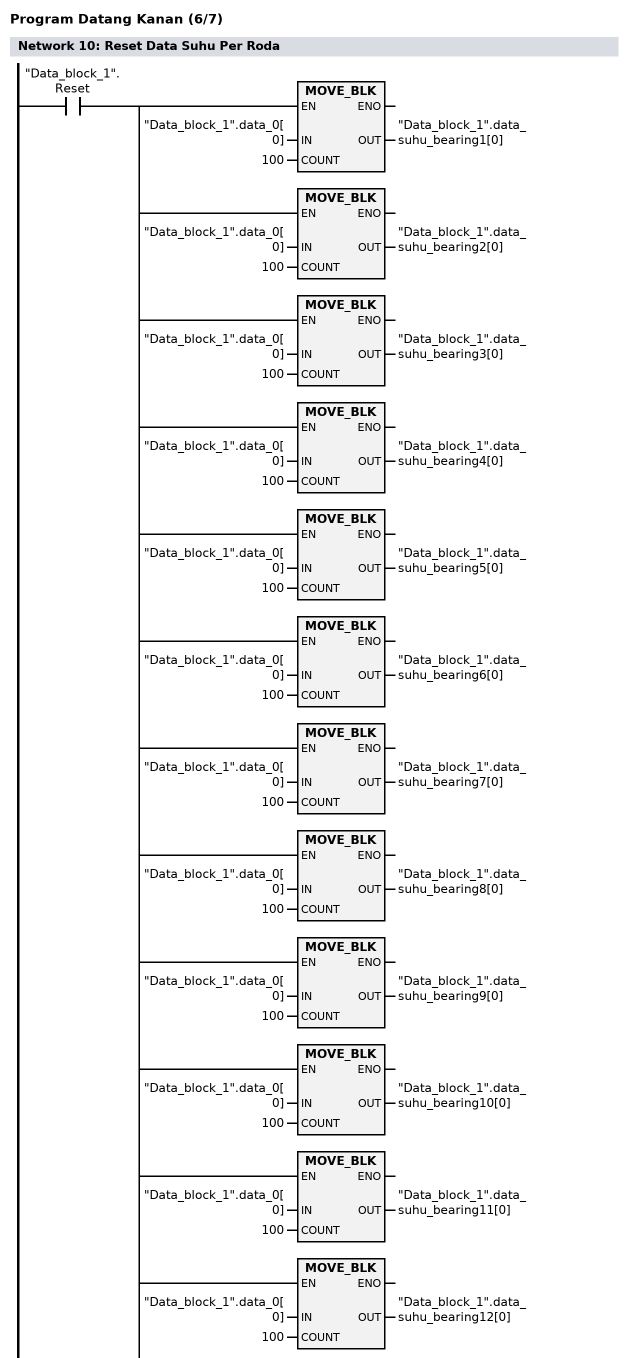
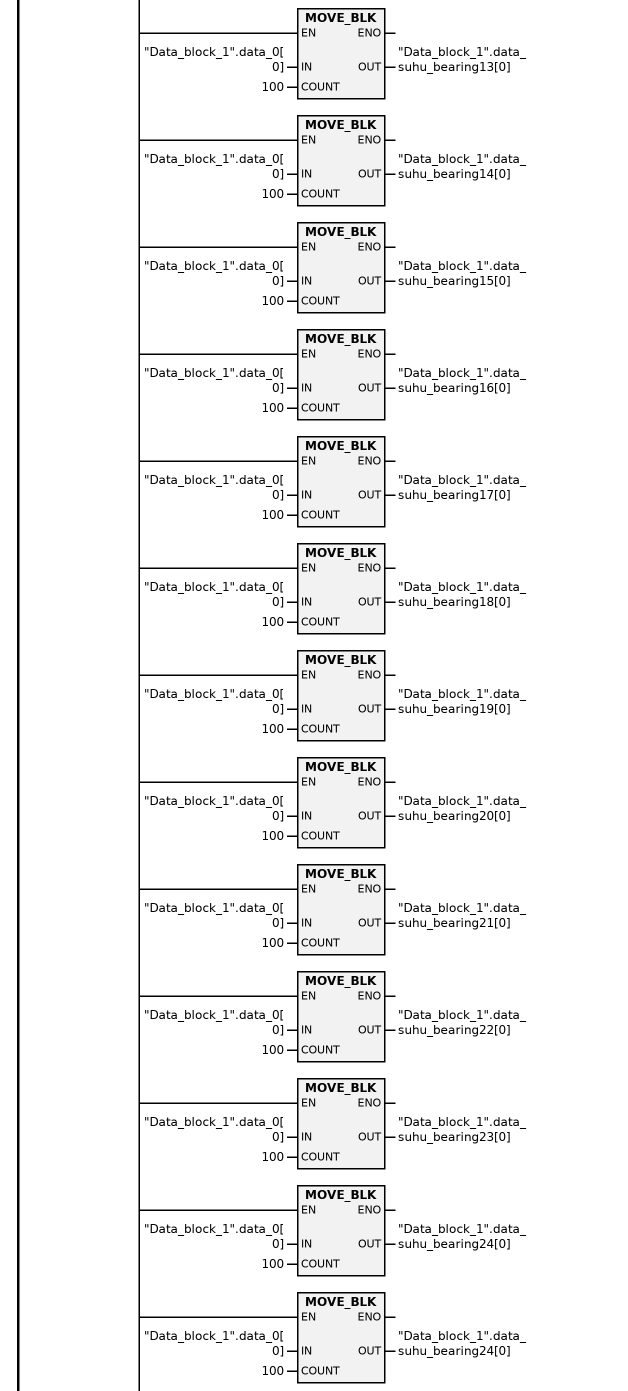
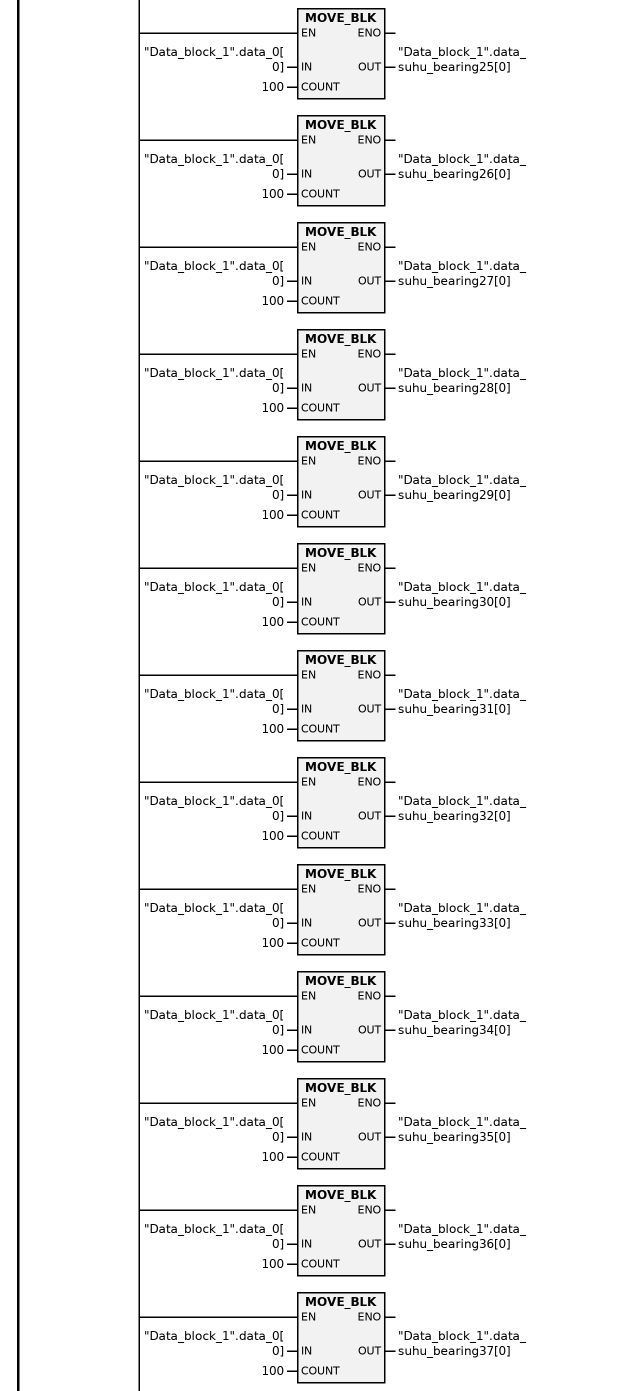
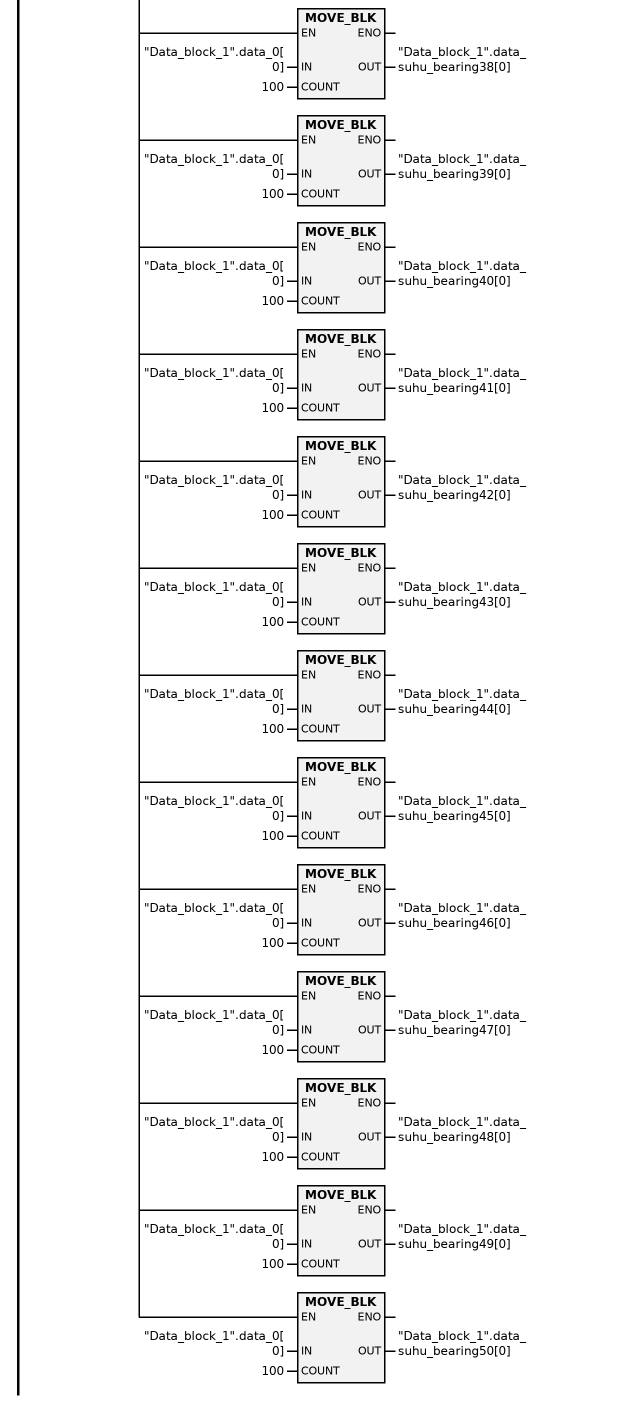
   #_w1 := "Data_block_1".Reset;
   IF #_w1 THEN
       MOVE_BLK(IN := "Data_block_1".data_0[0], COUNT := 100, OUT => "Data_block_1".data_suhu_bearing1[0]);
       MOVE_BLK(IN := "Data_block_1".data_0[0], COUNT := 100, OUT => "Data_block_1".data_suhu_bearing2[0]);
       MOVE_BLK(IN := "Data_block_1".data_0[0], COUNT := 100, OUT => "Data_block_1".data_suhu_bearing3[0]);
       MOVE_BLK(IN := "Data_block_1".data_0[0], COUNT := 100, OUT => "Data_block_1".data_suhu_bearing4[0]);
       MOVE_BLK(IN := "Data_block_1".data_0[0], COUNT := 100, OUT => "Data_block_1".data_suhu_bearing5[0]);
       MOVE_BLK(IN := "Data_block_1".data_0[0], COUNT := 100, OUT => "Data_block_1".data_suhu_bearing6[0]);
       MOVE_BLK(IN := "Data_block_1".data_0[0], COUNT := 100, OUT => "Data_block_1".data_suhu_bearing7[0]);
       MOVE_BLK(IN := "Data_block_1".data_0[0], COUNT := 100, OUT => "Data_block_1".data_suhu_bearing8[0]);
       MOVE_BLK(IN := "Data_block_1".data_0[0], COUNT := 100, OUT => "Data_block_1".data_suhu_bearing9[0]);
       MOVE_BLK(IN := "Data_block_1".data_0[0], COUNT := 100, OUT => "Data_block_1".data_suhu_bearing10[0]);
       MOVE_BLK(IN := "Data_block_1".data_0[0], COUNT := 100, OUT => "Data_block_1".data_suhu_bearing11[0]);
       MOVE_BLK(IN := "Data_block_1".data_0[0], COUNT := 100, OUT => "Data_block_1".data_suhu_bearing12[0]);
       MOVE_BLK(IN := "Data_block_1".data_0[0], COUNT := 100, OUT => "Data_block_1".data_suhu_bearing13[0]);
       MOVE_BLK(IN := "Data_block_1".data_0[0], COUNT := 100, OUT => "Data_block_1".data_suhu_bearing14[0]);
       MOVE_BLK(IN := "Data_block_1".data_0[0], COUNT := 100, OUT => "Data_block_1".data_suhu_bearing15[0]);
       MOVE_BLK(IN := "Data_block_1".data_0[0], COUNT := 100, OUT => "Data_block_1".data_suhu_bearing16[0]);
       MOVE_BLK(IN := "Data_block_1".data_0[0], COUNT := 100, OUT => "Data_block_1".data_suhu_bearing17[0]);
       MOVE_BLK(IN := "Data_block_1".data_0[0], COUNT := 100, OUT => "Data_block_1".data_suhu_bearing18[0]);
       MOVE_BLK(IN := "Data_block_1".data_0[0], COUNT := 100, OUT => "Data_block_1".data_suhu_bearing19[0]);
       MOVE_BLK(IN := "Data_block_1".data_0[0], COUNT := 100, OUT => "Data_block_1".data_suhu_bearing20[0]);
       MOVE_BLK(IN := "Data_block_1".data_0[0], COUNT := 100, OUT => "Data_block_1".data_suhu_bearing21[0]);
       MOVE_BLK(IN := "Data_block_1".data_0[0], COUNT := 100, OUT => "Data_block_1".data_suhu_bearing22[0]);
       MOVE_BLK(IN := "Data_block_1".data_0[0], COUNT := 100, OUT => "Data_block_1".data_suhu_bearing23[0]);
       MOVE_BLK(IN := "Data_block_1".data_0[0], COUNT := 100, OUT => "Data_block_1".data_suhu_bearing24[0]);
       MOVE_BLK(IN := "Data_block_1".data_0[0], COUNT := 100, OUT => "Data_block_1".data_suhu_bearing24[0]);
       MOVE_BLK(IN := "Data_block_1".data_0[0], COUNT := 100, OUT => "Data_block_1".data_suhu_bearing25[0]);
       MOVE_BLK(IN := "Data_block_1".data_0[0], COUNT := 100, OUT => "Data_block_1".data_suhu_bearing26[0]);
       MOVE_BLK(IN := "Data_block_1".data_0[0], COUNT := 100, OUT => "Data_block_1".data_suhu_bearing27[0]);
       MOVE_BLK(IN := "Data_block_1".data_0[0], COUNT := 100, OUT => "Data_block_1".data_suhu_bearing28[0]);
       MOVE_BLK(IN := "Data_block_1".data_0[0], COUNT := 100, OUT => "Data_block_1".data_suhu_bearing29[0]);
       MOVE_BLK(IN := "Data_block_1".data_0[0], COUNT := 100, OUT => "Data_block_1".data_suhu_bearing30[0]);
       MOVE_BLK(IN := "Data_block_1".data_0[0], COUNT := 100, OUT => "Data_block_1".data_suhu_bearing31[0]);
       MOVE_BLK(IN := "Data_block_1".data_0[0], COUNT := 100, OUT => "Data_block_1".data_suhu_bearing32[0]);
       MOVE_BLK(IN := "Data_block_1".data_0[0], COUNT := 100, OUT => "Data_block_1".data_suhu_bearing33[0]);
       MOVE_BLK(IN := "Data_block_1".data_0[0], COUNT := 100, OUT => "Data_block_1".data_suhu_bearing34[0]);
       MOVE_BLK(IN := "Data_block_1".data_0[0], COUNT := 100, OUT => "Data_block_1".data_suhu_bearing35[0]);
       MOVE_BLK(IN := "Data_block_1".data_0[0], COUNT := 100, OUT => "Data_block_1".data_suhu_bearing36[0]);
       MOVE_BLK(IN := "Data_block_1".data_0[0], COUNT := 100, OUT => "Data_block_1".data_suhu_bearing37[0]);
       MOVE_BLK(IN := "Data_block_1".data_0[0], COUNT := 100, OUT => "Data_block_1".data_suhu_bearing38[0]);
       MOVE_BLK(IN := "Data_block_1".data_0[0], COUNT := 100, OUT => "Data_block_1".data_suhu_bearing39[0]);
       MOVE_BLK(IN := "Data_block_1".data_0[0], COUNT := 100, OUT => "Data_block_1".data_suhu_bearing40[0]);
       MOVE_BLK(IN := "Data_block_1".data_0[0], COUNT := 100, OUT => "Data_block_1".data_suhu_bearing41[0]);
       MOVE_BLK(IN := "Data_block_1".data_0[0], COUNT := 100, OUT => "Data_block_1".data_suhu_bearing42[0]);
       MOVE_BLK(IN := "Data_block_1".data_0[0], COUNT := 100, OUT => "Data_block_1".data_suhu_bearing43[0]);
       MOVE_BLK(IN := "Data_block_1".data_0[0], COUNT := 100, OUT => "Data_block_1".data_suhu_bearing44[0]);
       MOVE_BLK(IN := "Data_block_1".data_0[0], COUNT := 100, OUT => "Data_block_1".data_suhu_bearing45[0]);
       MOVE_BLK(IN := "Data_block_1".data_0[0], COUNT := 100, OUT => "Data_block_1".data_suhu_bearing46[0]);
       MOVE_BLK(IN := "Data_block_1".data_0[0], COUNT := 100, OUT => "Data_block_1".data_suhu_bearing47[0]);
       MOVE_BLK(IN := "Data_block_1".data_0[0], COUNT := 100, OUT => "Data_block_1".data_suhu_bearing48[0]);
       MOVE_BLK(IN := "Data_block_1".data_0[0], COUNT := 100, OUT => "Data_block_1".data_suhu_bearing49[0]);
       MOVE_BLK(IN := "Data_block_1".data_0[0], COUNT := 100, OUT => "Data_block_1".data_suhu_bearing50[0]);
   END_IF;
END_REGION

REGION Network 11
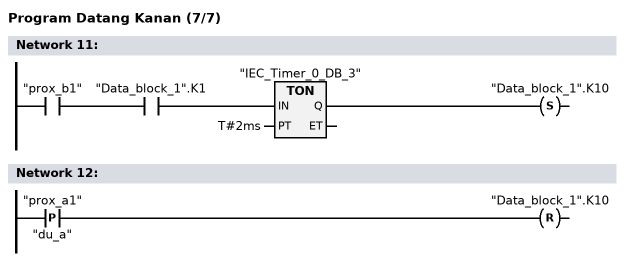
   "IEC_Timer_0_DB_3".TON(IN := "prox_b1" AND "Data_block_1".K1, PT := T#2ms);
   IF "IEC_Timer_0_DB_3".Q THEN "Data_block_1".K10 := TRUE; END_IF;
END_REGION

REGION Network 12
   RUNG wire#powerrail
      P_Contact(operand := "prox_a1", bit := "du_a")
      R_Coil( "Data_block_1".K10 )
   END_RUNG
   // the same network as SCL:
   #_w1 := "prox_a1" AND NOT "du_a";   // rising edge of "prox_a1"
   "du_a" := "prox_a1";
   IF #_w1 THEN "Data_block_1".K10 := FALSE; END_IF;
END_REGION
END_ORGANIZATION_BLOCK

ORGANIZATION_BLOCK "Program General"   // OB124, LAD, ProgramCycle
TITLE = General
{ S7_Optimized_Access := 'TRUE' }
VERSION : 0.1
   VAR_INPUT
      Initial_Call : Bool;   // Initial call of this OB
      Remanence : Bool;   // =True, if remanent data are available
   END_VAR
   VAR_TEMP   // added for the SCL form of the ladder/FBD networks
      _w1 : Bool;
   END_VAR
BEGIN

REGION Network 1: Counter sensor
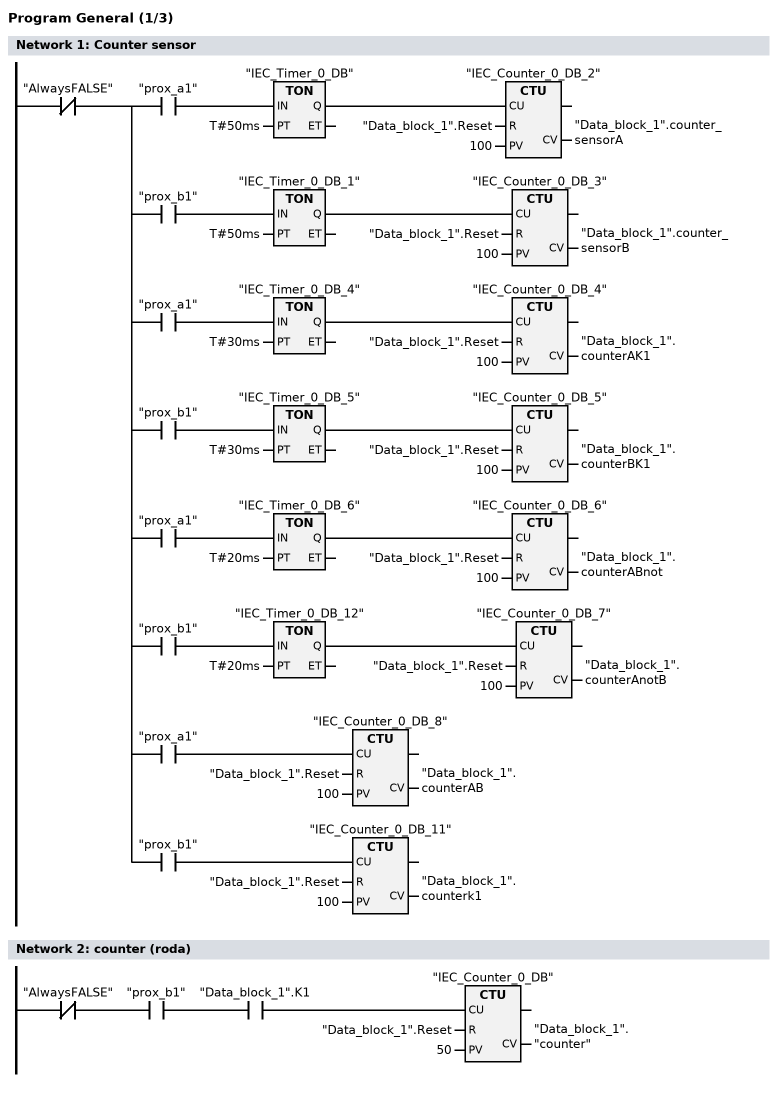
   "IEC_Timer_0_DB".TON(IN := NOT "AlwaysFALSE" AND "prox_a1", PT := T#50ms);
   "IEC_Counter_0_DB_2".CTU(CU := "IEC_Timer_0_DB".Q,
                           R := "Data_block_1".Reset,
                           PV := 100,
                           CV => "Data_block_1".counter_sensorA);
   "IEC_Timer_0_DB_1".TON(IN := NOT "AlwaysFALSE" AND "prox_b1", PT := T#50ms);
   "IEC_Counter_0_DB_3".CTU(CU := "IEC_Timer_0_DB_1".Q,
                           R := "Data_block_1".Reset,
                           PV := 100,
                           CV => "Data_block_1".counter_sensorB);
   "IEC_Timer_0_DB_4".TON(IN := NOT "AlwaysFALSE" AND "prox_a1", PT := T#30ms);
   "IEC_Counter_0_DB_4".CTU(CU := "IEC_Timer_0_DB_4".Q,
                           R := "Data_block_1".Reset,
                           PV := 100,
                           CV => "Data_block_1".counterAK1);
   "IEC_Timer_0_DB_5".TON(IN := NOT "AlwaysFALSE" AND "prox_b1", PT := T#30ms);
   "IEC_Counter_0_DB_5".CTU(CU := "IEC_Timer_0_DB_5".Q,
                           R := "Data_block_1".Reset,
                           PV := 100,
                           CV => "Data_block_1".counterBK1);
   "IEC_Timer_0_DB_6".TON(IN := NOT "AlwaysFALSE" AND "prox_a1", PT := T#20ms);
   "IEC_Counter_0_DB_6".CTU(CU := "IEC_Timer_0_DB_6".Q,
                           R := "Data_block_1".Reset,
                           PV := 100,
                           CV => "Data_block_1".counterABnot);
   "IEC_Timer_0_DB_12".TON(IN := NOT "AlwaysFALSE" AND "prox_b1", PT := T#20ms);
   "IEC_Counter_0_DB_7".CTU(CU := "IEC_Timer_0_DB_12".Q,
                           R := "Data_block_1".Reset,
                           PV := 100,
                           CV => "Data_block_1".counterAnotB);
   "IEC_Counter_0_DB_8".CTU(CU := NOT "AlwaysFALSE" AND "prox_a1",
                           R := "Data_block_1".Reset,
                           PV := 100,
                           CV => "Data_block_1".counterAB);
   "IEC_Counter_0_DB_11".CTU(CU := NOT "AlwaysFALSE" AND "prox_b1",
                           R := "Data_block_1".Reset,
                           PV := 100,
                           CV => "Data_block_1".counterk1);
END_REGION

REGION Network 2: counter (roda)
   "IEC_Counter_0_DB".CTU(CU := NOT "AlwaysFALSE" AND "prox_b1" AND "Data_block_1".K1,
                          R := "Data_block_1".Reset,
                          PV := 50,
                          CV => "Data_block_1"."counter");
END_REGION

REGION Network 3: Timer Mengukur kecepatan kereta
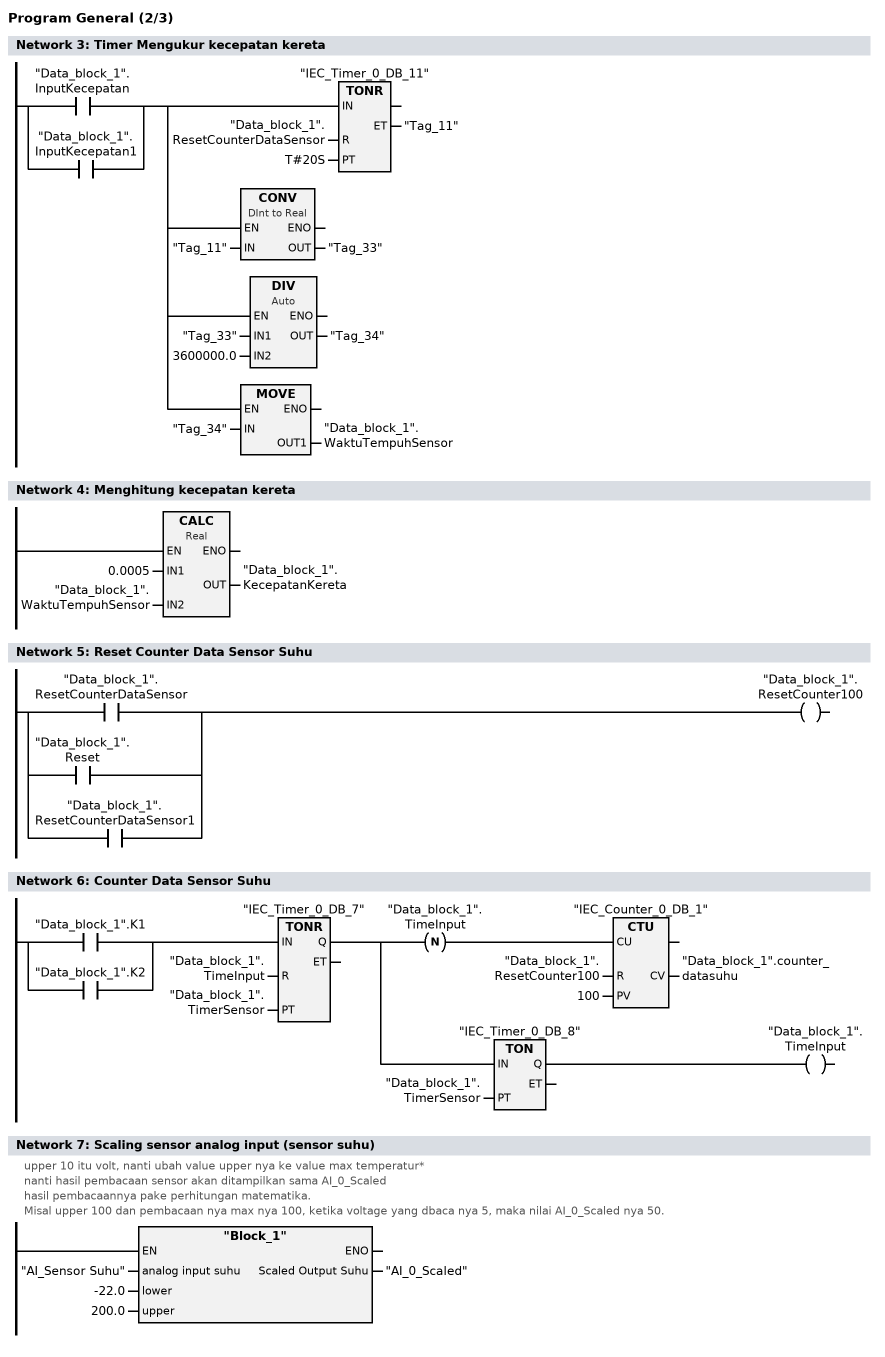
   #_w1 := "Data_block_1".InputKecepatan OR "Data_block_1".InputKecepatan1;
   "IEC_Timer_0_DB_11".TONR(IN := #_w1, R := "Data_block_1".ResetCounterDataSensor, PT := T#20S, ET => "Tag_11");
   IF #_w1 THEN
       "Tag_33" := DINT_TO_REAL("Tag_11");
       "Tag_34" := "Tag_33" / 3600000.0;
       "Data_block_1".WaktuTempuhSensor := "Tag_34";
   END_IF;
END_REGION

REGION Network 4: Menghitung kecepatan kereta
   CALC(in1 := 0.0005, in2 := "Data_block_1".WaktuTempuhSensor, out => "Data_block_1".KecepatanKereta);
END_REGION

REGION Network 5: Reset Counter Data Sensor Suhu
   RUNG wire#powerrail
      Contact( "Data_block_1".ResetCounterDataSensor )
      wire#w1
      Coil( "Data_block_1".ResetCounter100 )
   END_RUNG
   RUNG wire#powerrail
      Contact( "Data_block_1".Reset )
   END_RUNG wire#w1
   RUNG wire#powerrail
      Contact( "Data_block_1".ResetCounterDataSensor1 )
   END_RUNG wire#w1
   // the same network as SCL:
   "Data_block_1".ResetCounter100 := "Data_block_1".ResetCounterDataSensor OR "Data_block_1".Reset OR "Data_block_1".ResetCounterDataSensor1;
END_REGION

REGION Network 6: Counter Data Sensor Suhu
   "IEC_Timer_0_DB_7".TONR(IN := "Data_block_1".K1 OR "Data_block_1".K2,
                           R := "Data_block_1".TimeInput,
                           PT := "Data_block_1".TimerSensor);
   #_w1 := NOT "IEC_Timer_0_DB_7".Q AND "Data_block_1".TimeInput;   // falling edge
   "Data_block_1".TimeInput := "IEC_Timer_0_DB_7".Q;
   "IEC_Counter_0_DB_1".CTU(CU := #_w1,
                           R := "Data_block_1".ResetCounter100,
                           PV := 100,
                           CV => "Data_block_1".counter_datasuhu);
   "IEC_Timer_0_DB_8".TON(IN := "IEC_Timer_0_DB_7".Q, PT := "Data_block_1".TimerSensor);
   "Data_block_1".TimeInput := "IEC_Timer_0_DB_8".Q;
END_REGION

REGION Network 7: Scaling sensor analog input (sensor suhu)
   // upper 10 itu volt, nanti ubah value upper nya ke value max temperatur* 
   // nanti hasil pembacaan sensor akan ditampilkan sama AI_0_Scaled
   // hasil pembacaannya pake perhitungan matematika. 
   // Misal upper 100 dan pembacaan nya max nya 100, ketika voltage yang dbaca nya 5, maka nilai AI_0_Scaled nya 50.
   RUNG wire#powerrail
      "Block_1"("analog input suhu" := "AI_Sensor Suhu", lower := -22.0, upper := 200.0, "Scaled Output Suhu" => "AI_0_Scaled")
   END_RUNG
   // the same network as SCL:
   "Block_1"("analog input suhu" := "AI_Sensor Suhu",
             lower := -22.0,
             upper := 200.0,
             "Scaled Output Suhu" => "AI_0_Scaled");
END_REGION

REGION Network 8: Data memory suhu kanan
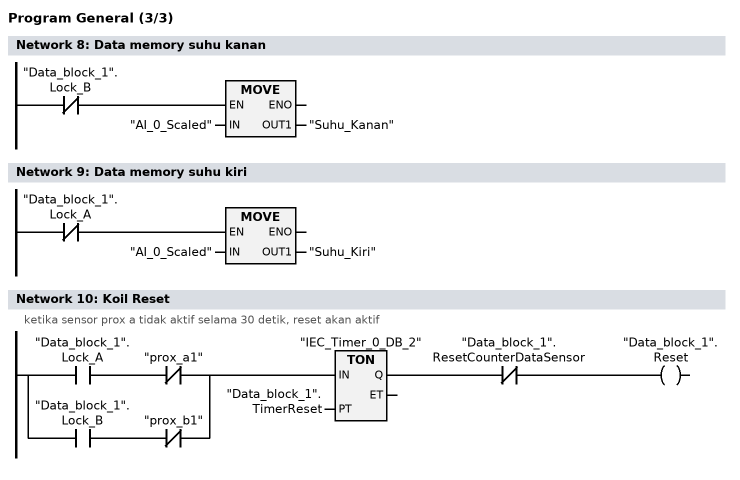
   RUNG wire#powerrail
      I_Contact( "Data_block_1".Lock_B )
      Move(in := "AI_0_Scaled", out1 => "Suhu_Kanan")
   END_RUNG
   // the same network as SCL:
   IF NOT "Data_block_1".Lock_B THEN "Suhu_Kanan" := "AI_0_Scaled"; END_IF;
END_REGION

REGION Network 9: Data memory suhu kiri
   RUNG wire#powerrail
      I_Contact( "Data_block_1".Lock_A )
      Move(in := "AI_0_Scaled", out1 => "Suhu_Kiri")
   END_RUNG
   // the same network as SCL:
   IF NOT "Data_block_1".Lock_A THEN "Suhu_Kiri" := "AI_0_Scaled"; END_IF;
END_REGION

REGION Network 10: Koil Reset
   // ketika sensor prox a tidak aktif selama 30 detik, reset akan aktif
   "IEC_Timer_0_DB_2".TON(IN := ("Data_block_1".Lock_A AND NOT "prox_a1") OR ("Data_block_1".Lock_B AND NOT "prox_b1"),
                          PT := "Data_block_1".TimerReset);
   "Data_block_1".Reset := "IEC_Timer_0_DB_2".Q AND NOT "Data_block_1".ResetCounterDataSensor;
END_REGION
END_ORGANIZATION_BLOCK

(* ===== HMI "HMI_RT_1" =====
system functions are stored by id; their names below are inferred from use
connection "Connection_1": ETHERNET, S7_1200_OMS
connection "HMI_Connection_1": ETHERNET, S7_1200_OMS

HMI tags "Default tag table"
   "prox_a" : Bool = PLC prox_a1 AT %I0.0, 1 s
   "prox_b" : Bool = PLC prox_b1 AT %I0.1, 1 s
   "Q1" : Bool = PLC "Q1-1" AT %M0.0, 1 s
   "Q2" : Bool = PLC "Q2-1" AT %M0.1, 1 s
   "du_a" : Bool = PLC du_a AT %M0.2, 1 s
   "dd_b" : Bool = PLC dd_b AT %M0.3, 1 s
   "k_proxa" : Bool = PLC k_proxa AT %M0.4, 1 s
   "k_proxb" : Bool = PLC k_proxb AT %M0.5, 1 s
   "counter" : Bool = PLC counter AT %M0.6, 1 s
   "pemutus" : Bool = PLC pemutus AT %M0.7, 1 s
   "du_b" : Bool = PLC "ProxA+" AT %M1.0, 1 s
   "dd_a" : Bool = PLC "ProxB-" AT %M1.1, 1 s
   "reset" : Bool = PLC reset AT %M1.2, 1 s
   "Clock_Byte" : Byte = PLC Clock_Byte AT %MB10, 1 s
   "Clock_10Hz" : Bool = PLC Clock_10Hz AT %M10.0, 1 s
   "Clock_5Hz" : Bool = PLC Clock_5Hz AT %M10.1, 1 s
   "Clock_2.5Hz" : Bool = PLC "Clock_2.5Hz" AT %M10.2, 1 s
   "Clock_2Hz" : Bool = PLC Clock_2Hz AT %M10.3, 1 s
   "Clock_1.25Hz" : Bool = PLC "Clock_1.25Hz" AT %M10.4, 1 s
   "Clock_1Hz" : Bool = PLC Clock_1Hz AT %M10.5, 1 s
   "Clock_0.625Hz" : Bool = PLC "Clock_0.625Hz" AT %M10.6, 1 s
   "Clock_0.5Hz" : Bool = PLC "Clock_0.5Hz" AT %M10.7, 1 s
   "System_Byte" : Byte = PLC System_Byte AT %MB100, 1 s
   "FirstScan" : Bool = PLC FirstScan AT %M100.0, 1 s
   "DiagStatusUpdate" : Bool = PLC DiagStatusUpdate AT %M100.1, 1 s
   "AlwaysTRUE" : Bool = PLC AlwaysTRUE AT %M100.2, 1 s
   "AlwaysFALSE" : Bool = PLC AlwaysFALSE AT %M100.3, 1 s
   "Data_block_1_dataroda1{0}" : Real = PLC Data_block_1.dataroda1[0] AT %DB3.DBD21370, 1 s
   "Data_block_1_dataroda1{1}" : Real = PLC Data_block_1.dataroda1[1] AT %DB3.DBD21374, 1 s
   "Data_block_1_dataroda1{2}" : Real = PLC Data_block_1.dataroda1[2] AT %DB3.DBD21378, 1 s
   "Data_block_1_dataroda1{3}" : Real = PLC Data_block_1.dataroda1[3] AT %DB3.DBD21382, 1 s

screen "Screen_1" 1024x768
   on GenerateScreen: function_bb0abc73()
   Switch "Switch_1" at 110,0 size 120x88; CaptionText 'a'; TextOff 'OFF'; TextOn 'ON'
      ProcessValue <- "prox_a"
   Switch "Switch_2" at 256,0 size 120x88; CaptionText 'b'; TextOff 'OFF'; TextOn 'ON'
      ProcessValue <- "prox_b"
   StatusForce "Watch table_1" at 49,111 size 600x300; ToolTipText 'Text'
*)